// TIA Portal project "ARDOUINOS7" (V15)

(* hardware
DEVICE "S7-1200 station_1"  S7-1200 Station
   slot 0: "Rack_0"  S7-1200 Rack  Rack  V1.0
   slot 1: "PLC_1"  CPU 1214C DC/DC/DC  6ES7 214-1AG40-0XB0  V4.1
DEVICE "PC-System_1"  SIMATIC PC station
   slot 0: "SIMATIC PC station"  Rail  SIMATIC PC-Station  V1.0
      slot 125: "Stationmanager"  Station_Manager  V6.0.4
   slot 1: "HMI_RT_1"  WinCC RT Advanced  6AV2 104-0xxxx-xxxx  15.0.0.0
      slot 33792: "Host interface"  Host interface
   slot 2: "IE general_1"  IE General  IE_CP  V8.2.0
*)

// ===== PLC "PLC_1"  CPU 1214C DC/DC/DC =====

DATA_BLOCK "Data_block_1"   // DB2
{ S7_Optimized_Access := 'FALSE' }
VERSION : 0.1
   VAR
      Ready : Bool;
      courant : Int;
      in_use : Bool;
      freaquance : Int;
      thermostor : Bool;
      vitesse : Int;
      defaut : Bool;
      Mfreaquance : Int;
      S3 : Bool;
      S4 : Bool;
      distance : Int;
      pompep60 : Bool;
      "time" : Int;
      pompeRege : Bool;
      time2 : Int;
      pipe : Bool;
      "20hz" : Bool;
      "30hz" : Bool;
      "40hz" : Bool;
   END_VAR
BEGIN
END_DATA_BLOCK

ORGANIZATION_BLOCK "Main"   // OB1, LAD, ProgramCycle
TITLE = "Main Program Sweep (Cycle)"
{ S7_Optimized_Access := 'TRUE' }
VERSION : 0.1
   VAR_INPUT
      Initial_Call : Bool;   // Initial call of this OB
      Remanence : Bool;   // =True, if remanent data are available
   END_VAR
BEGIN

REGION Network 1: pipe&constsant_speed
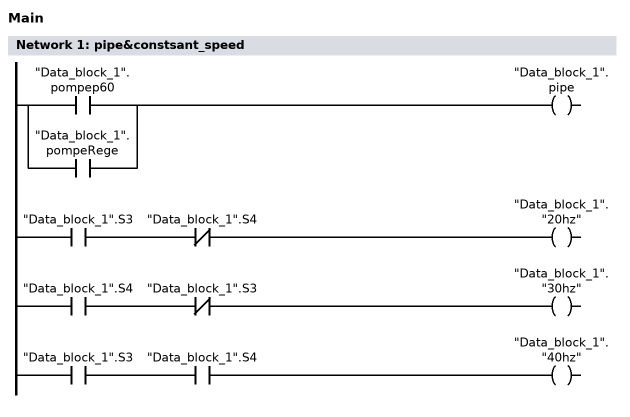
   RUNG wire#powerrail
      Contact( "Data_block_1".pompep60 )
      wire#w1
      Coil( "Data_block_1".pipe )
   END_RUNG
   RUNG wire#powerrail
      Contact( "Data_block_1".pompeRege )
   END_RUNG wire#w1
   RUNG wire#powerrail
      Contact( "Data_block_1".S3 )
      I_Contact( "Data_block_1".S4 )
      Coil( "Data_block_1"."20hz" )
   END_RUNG
   RUNG wire#powerrail
      Contact( "Data_block_1".S4 )
      I_Contact( "Data_block_1".S3 )
      Coil( "Data_block_1"."30hz" )
   END_RUNG
   RUNG wire#powerrail
      Contact( "Data_block_1".S3 )
      Contact( "Data_block_1".S4 )
      Coil( "Data_block_1"."40hz" )
   END_RUNG
   // the same network as SCL:
   "Data_block_1".pipe := "Data_block_1".pompep60 OR "Data_block_1".pompeRege;
   "Data_block_1"."20hz" := "Data_block_1".S3 AND NOT "Data_block_1".S4;
   "Data_block_1"."30hz" := "Data_block_1".S4 AND NOT "Data_block_1".S3;
   "Data_block_1"."40hz" := "Data_block_1".S3 AND "Data_block_1".S4;
END_REGION
END_ORGANIZATION_BLOCK

(* ===== HMI "HMI_RT_1" =====
system functions are stored by id; their names below are inferred from use
connection "HMI_Connection_1": ETHERNET, S7_1200_OMS

HMI tags "Default tag table"
   "Data_block_1_ready" : Bool = PLC Data_block_1.Ready AT %DB2.DBX0.0, 1 s
   "Data_block_1_pompeRege" : Bool = PLC Data_block_1.pompeRege AT %DB2.DBX24.0, 1 s
   "Data_block_1_freaquance" : Int = PLC Data_block_1.freaquance AT %DB2.DBW6, 1 s
   "Data_block_1_distance" : Int = PLC Data_block_1.distance AT %DB2.DBW18, 1 s
   "Data_block_1_Mfreaquance" : Int = PLC Data_block_1.Mfreaquance AT %DB2.DBW14, 1 s
   "Data_block_1_pompep60" : Bool = PLC Data_block_1.pompep60 AT %DB2.DBX20.0, 1 s
   "Data_block_1_S3" : Bool = PLC Data_block_1.S3 AT %DB2.DBX16.0, 1 s
   "Data_block_1_S4" : Bool = PLC Data_block_1.S4 AT %DB2.DBX16.1, 1 s
   "Data_block_1_in_use" : Bool = PLC Data_block_1.in_use AT %DB2.DBX4.0, 1 s
   "Data_block_1_thermostor" : Bool = PLC Data_block_1.thermostor AT %DB2.DBX8.0, 1 s
   "Data_block_1_defaut" : Bool = PLC Data_block_1.defaut AT %DB2.DBX12.0, 1 s
   "Data_block_1_vitesse" : Int = PLC Data_block_1.vitesse AT %DB2.DBW10, 1 s
   "Data_block_1_courant" : Int = PLC Data_block_1.courant AT %DB2.DBW2, 1 s
   "Data_block_1_pipe" : Bool = PLC Data_block_1.pipe AT %DB2.DBX28.0, 1 s
   "Data_block_1_20hz" : Bool = PLC Data_block_1.20hz AT %DB2.DBX28.1, 1 s
   "Data_block_1_30hz" : Bool = PLC Data_block_1.30hz AT %DB2.DBX28.2, 1 s
   "Data_block_1_40hz" : Bool = PLC Data_block_1.40hz AT %DB2.DBX28.3, 1 s

text list "MfreaquanceVal": 15 '15 Hz'; 16 '16 Hz'; 17 '17 Hz'; 18 '18 Hz'; 19 '19 Hz'; 20 '20 Hz'; 21 '21 Hz'; 22 '22 Hz'; 23 '23 Hz'; 24 '24 Hz'; 25 '25 Hz'; 26 '26 Hz'; 27 '27 Hz'; 28 '28 Hz'; 29 '29 Hz'; 30 '30 Hz'; 31 '31 Hz'; 32 '32 Hz'; 33 '33 Hz'; 34 '34 Hz'; 35 '35 Hz'; 36 '36 Hz'; 37 '37 Hz'; 38 '38 Hz'; 39 '39 Hz'; 40 '40 Hz'; 41 '41 Hz'; 42 '42 Hz'; 43 '43 Hz'; 44 '44 Hz'; 45 '45 Hz'; 46 '46 Hz'; 47 '47 Hz'; 48 '48 Hz'; 49 '49 Hz'; 50 '50 Hz'

screen "Screen_1" 1024x768
   SymbolLibrary "Symbol library_3" at 406,441 size 86x55
      ProcessValue <- "Data_block_1_pompeRege"
      Appearance <- "Data_block_1_pipe"
   SymbolLibrary "Symbol library_4" at 232,441 size 176x28
      Appearance <- "Data_block_1_pompeRege"
   SymbolLibrary "Symbol library_5" at 177,441 size 57x54
      Appearance <- "Data_block_1_pompeRege"
   SymbolLibrary "Symbol library_6" at 675,441 size 69x54
      Appearance <- "Data_block_1_pompep60"
   SymbolLibrary "Symbol library_7" at 427,495 size 44x272
      Appearance <- "Data_block_1_pipe"
   SymbolLibrary "Symbol library_9" at 490,441 size 186x28
      Appearance <- "Data_block_1_pompep60"
   SymbolLibrary "Symbol library_10" at 709,479 size 34x120
      ProcessValue <- "Data_block_1_pompep60"
      Appearance <- "Data_block_1_pompep60"
   SymbolLibrary "Symbol library_12" at 175,495 size 33x28
      Appearance <- "Data_block_1_pompeRege"
   Bar "niveaux" at 613,530 size 363x230; Unit Cm; MinimumValue 0; MaximumValue 200
      ProcessValue <- "Data_block_1_distance"
   SymbolLibrary "Symbol library_2" at 5,522 size 224x120
      ProcessValue <- "Data_block_1_pompeRege"
      Appearance <- "Data_block_1_pompeRege"
   SymbolLibrary "Symbol library_13" at 227,572 size 53x57
      Appearance <- "Data_block_1_pompeRege"
   IOField "I/O field_1" at 526,319 size 60x32; FormatPattern 99; Unit  Hz
      ProcessValue <- "Data_block_1_freaquance"
   IOField "I/O field_2" at 908,319 size 58x32; FormatPattern 99; Unit  A
      ProcessValue <- "Data_block_1_courant"
   IOField "I/O field_3" at 688,319 size 112x32; FormatPattern 9999; Unit  Tr/Min
      ProcessValue <- "Data_block_1_vitesse"
   Button "Button_9" at 499,72 size 96x32; TextOff 'Ready'
      on Click: SetBit("Data_block_1_S4"); ResetBit("Data_block_1_S3")
      Appearance <- "Data_block_1_ready"
   Button "Button_7" at 624,75 size 96x32; TextOff 'En Marche'
      on Click: SetBit("Data_block_1_S4"); ResetBit("Data_block_1_S3")
      Appearance <- "Data_block_1_in_use"
   Button "Button_6" at 750,76 size 96x32; TextOff 'Thermostor'
      on Click: SetBit("Data_block_1_S3"); ResetBit("Data_block_1_S4")
      Appearance <- "Data_block_1_thermostor"
   Button "Button_8" at 880,80 size 96x32; TextOff 'Defaut'
      on Click: SetBit("Data_block_1_S3"); SetBit("Data_block_1_S4")
      Appearance <- "Data_block_1_defaut"
   Slider "Slider_1" at 163,93 size 80x219; Caption 'Frequance'
      ProcessValue <- "Data_block_1_Mfreaquance"
   Gauge "Gauge_1" at 483,155 size 147x147; CaptionText 'Frequance P60'; UnitText 'Hz'
      ProcessValue <- "Data_block_1_freaquance"
   Button "Button_2" at 15,64 size 148x40; TextOff 'Pompe P60'
      Appearance <- "Data_block_1_pompep60"
   Gauge "Gauge_2" at 653,120 size 182x182; UnitText 'Tr/Min'; CaptionText 'Vitesse pP60'
      ProcessValue <- "Data_block_1_vitesse"
   Gauge "Gauge_3" at 863,155 size 147x147; UnitText 'A'; CaptionText 'Courant P60'
      ProcessValue <- "Data_block_1_courant"
   Switch "Switch_2" at 16,104 size 120x59; TextOn 'Demaré'; CaptionText 'Pompe P60'; TextOff 'Arreté'
      ProcessValue <- "Data_block_1_pompep60"
      on SwitchOff: ResetBit("Data_block_1_S3"); ResetBit("Data_block_1_S4")
   Button "Button_3" at 15,185 size 96x32; TextOff '20 Hz'
      on Click: SetBit("Data_block_1_S3"); ResetBit("Data_block_1_S4")
      Appearance <- "Data_block_1_20hz"
   Button "Button_4" at 16,245 size 96x32; TextOff '30 Hz'
      on Click: SetBit("Data_block_1_S4"); ResetBit("Data_block_1_S3")
      Appearance <- "Data_block_1_30hz"
   Button "Button_5" at 15,302 size 96x32; TextOff '40 Hz'
      on Click: SetBit("Data_block_1_S3"); SetBit("Data_block_1_S4")
      Appearance <- "Data_block_1_40hz"
   Button "Button_1" at 299,67 size 148x40; TextOff 'Pompe Rege'
      Appearance <- "Data_block_1_pompeRege"
   Switch "Switch_1" at 325,108 size 120x59; CaptionText 'Pompe Rege'; TextOff 'Arreté'; TextOn 'Demaré'
      ProcessValue <- "Data_block_1_pompeRege"
   SymbolLibrary "Symbol library_1" at 719,408 size 138x291
      ProcessValue <- "Data_block_1_pompep60"
      Appearance <- "Data_block_1_pompep60"
   SymbolLibrary "Symbol library_14" at 253,620 size 27x120
      Appearance <- "Data_block_1_pompeRege"
   SymbolicIOField "Symbolic I/O field_1" at 163,316 size 92x32; TextOff '0'; TextOn '1'; TextList "MfreaquanceVal"
      ProcessValue <- "Data_block_1_Mfreaquance"
   TextField "Text field_1" at 631,13 size 201x28; Text 'Etas Du Pompe P60'
   TextField "Text field_2" at 24,13 size 399x28; Text 'Controle Du Pompe P60 & Pompe Regé'
*)